{attribute 'pack_mode' := '2'}
TYPE ST_DATA_CTRL :
STRUCT
  Cmd       : E_DATA_CTRL;
END_STRUCT
END_TYPE

(* stored: Version 1.1.0.1, ProductVersion 3.1.4026.18
   DUT ST_DATA_CTRL: Id {67c50860-e659-4b76-8476-f836b9442076} *)
